(* IEC 61131-3 sources: RL_MAR/experiments/comparison/autoplc/results/deepseek-ai-DeepSeek-V3.2_20260508_111905/med_29, 1 file *)

(* ---- med_29_1.st ---- *)
FUNCTION_BLOCK DocumentFilingSystem
VAR_INPUT
    DocumentInlet : BOOL; (* Input to detect the arrival of a document *)
    CategorySelector : INT; (* Input to select the document category *)
END_VAR
VAR_OUTPUT
    ConveyorMotor : BOOL; (* Output to control the conveyor motor *)
    StorageBin1 : BOOL; (* Output to activate storage bin 1 *)
    StorageBin2 : BOOL; (* Output to activate storage bin 2 *)
    StorageBin3 : BOOL; (* Output to activate storage bin 3 *)
    StorageBin4 : BOOL; (* Output to activate storage bin 4 *)
END_VAR

VAR
    // Internal variables for state management
    bProcessingCondition : BOOL;
    bValidCategory : BOOL;
END_VAR

(* Main control logic *)
(* Initialize outputs *)
ConveyorMotor := FALSE;
StorageBin1 := FALSE;
StorageBin2 := FALSE;
StorageBin3 := FALSE;
StorageBin4 := FALSE;

(* Check if category is valid (1-4) *)
bValidCategory := (CategorySelector >= 1) AND (CategorySelector <= 4);

(* Determine if processing conditions are met *)
bProcessingCondition := DocumentInlet AND bValidCategory;

(* Process based on conditions *)
IF bProcessingCondition THEN
    (* Activate conveyor motor *)
    ConveyorMotor := TRUE;

    (* Activate appropriate storage bin based on category *)
    CASE CategorySelector OF
        1:
            StorageBin1 := TRUE;
            StorageBin2 := FALSE;
            StorageBin3 := FALSE;
            StorageBin4 := FALSE;
        2:
            StorageBin1 := FALSE;
            StorageBin2 := TRUE;
            StorageBin3 := FALSE;
            StorageBin4 := FALSE;
        3:
            StorageBin1 := FALSE;
            StorageBin2 := FALSE;
            StorageBin3 := TRUE;
            StorageBin4 := FALSE;
        4:
            StorageBin1 := FALSE;
            StorageBin2 := FALSE;
            StorageBin3 := FALSE;
            StorageBin4 := TRUE;
    END_CASE;
ELSE
    (* Deactivate all outputs when no document or invalid category *)
    ConveyorMotor := FALSE;
    StorageBin1 := FALSE;
    StorageBin2 := FALSE;
    StorageBin3 := FALSE;
    StorageBin4 := FALSE;
END_IF;

END_FUNCTION_BLOCK
